FUNCTION_BLOCK T_ResultAggregate IMPLEMENTS I_ExecutionResult
VAR
	Results : ARRAY[0..ResultsUpperBound] OF I_ExecutionResult;
	Count   : UINT;
END_VAR
VAR CONSTANT
	ResultsUpperBound : UINT := 99;
END_VAR

METHOD Abort
VAR
    i      : DINT;
    Result : I_ExecutionResult;
    IP     : I_ListItem;
END_VAR
IF Count > 0 THEN
	FOR i := 0 TO Count - 1 DO
		Result := Results[i];
		IF Result <> 0 THEN
            Result.Abort(); 
        END_IF
    END_FOR
END_IF
END_METHOD

PROPERTY Aborted : BOOL
GET
VAR
    i      : UINT;
    Result : I_ExecutionResult;
END_VAR
Aborted := TRUE;
IF Count > 0 THEN
	FOR i := 0 TO Count - 1 DO
		Result := Results[i];
		IF Result <> 0 THEN
			Aborted := Aborted AND Result.Aborted; // Done if all result.aborted
		END_IF
	END_FOR
END_IF
END_GET
END_PROPERTY

PROPERTY Aborting : BOOL
GET
VAR
    i      : DINT;
    Result : I_ExecutionResult;
    IP     : I_ListItem;
END_VAR
Aborting := FALSE;
IF Count > 0 THEN
	FOR i := 0 TO Count - 1 DO
		Result := Results[i];
		IF Result <> 0 THEN
            Aborting := Aborting OR Result.Aborting; // Busy if any result.aborting
        END_IF
    END_FOR
END_IF
END_GET
END_PROPERTY

METHOD AddResult : BOOL
VAR_INPUT
	Result : I_ExecutionResult;
END_VAR
IF Count <= ResultsUpperBound THEN
	Results[Count] := Result;
	F_Inc(Count);
	AddResult := TRUE;
END_IF
END_METHOD

PROPERTY Busy : BOOL
GET
VAR
    i      : DINT;
    Result : I_ExecutionResult;
    IP     : I_ListItem;
END_VAR
Busy := FALSE;
IF Count > 0 THEN
	FOR i := 0 TO Count - 1 DO
		Result := Results[i];
		IF Result <> 0 THEN
            Busy := Busy OR Result.Busy; // Busy if any result.busy
        END_IF
    END_FOR
END_IF
END_GET
END_PROPERTY

METHOD Clear
VAR
    i      : UINT;
    Result : I_ExecutionResult;
END_VAR
IF Count > 0 THEN
    FOR i := 0 TO Count - 1 DO
		Result := Results[i];
		IF Result <> 0 THEN
			Result.Clear(); 
		END_IF
	END_FOR
END_IF

F_ClearMem(Results);
Count := 0;
END_METHOD

PROPERTY Done : BOOL
GET
VAR
    i      : DINT;
    Result : I_ExecutionResult;
    IP     : I_ListItem;
END_VAR
Done := TRUE;
IF Count > 0 THEN
	FOR i := 0 TO Count - 1 DO
		Result := Results[i];
		IF Result <> 0 THEN
			Done := Done AND Result.Done; // Done if all result.done
		END_IF
	END_FOR
END_IF
END_GET
END_PROPERTY

PROPERTY Error : BOOL
GET
VAR
    i      : DINT;
    Result : I_ExecutionResult;
    IP     : I_ListItem;
END_VAR
Error := FALSE;
IF Count > 0 THEN
	FOR i := 0 TO Count - 1 DO
		Result := Results[i];
		IF Result <> 0 THEN
			Error := Error OR Result.Error; // Error if any result.error
		END_IF
	END_FOR
END_IF
END_GET
END_PROPERTY

PROPERTY ErrorMsg : Tc2_System.T_MaxString
GET
VAR
    i      : DINT;
    Result : I_ExecutionResult;
    IP     : I_ListItem;
END_VAR
ErrorMsg := '';
IF Count > 0 THEN
	FOR i := 0 TO Count - 1 DO
		Result := Results[i];
		IF Result <> 0 THEN
			IF Result.Error THEN
				ErrorMsg := Result.ErrorMsg;
				RETURN;
			END_IF
		END_IF
	END_FOR
END_IF
END_GET
END_PROPERTY

PROPERTY Ready : BOOL
GET
VAR
    i      : DINT;
    Result : I_ExecutionResult;
    IP     : I_ListItem;
END_VAR
Ready := TRUE;
IF Count > 0 THEN
	FOR i := 0 TO Count - 1 DO
		Result := Results[i];
		IF Result <> 0 THEN
            Ready := Ready AND Result.Ready; // Ready if all result.ready
        END_IF
    END_FOR
END_IF
END_GET
END_PROPERTY

PROPERTY ResultCount : DINT
GET
ResultCount := Count;
END_GET
END_PROPERTY

PROPERTY Starting : BOOL
GET
VAR
    i      : DINT;
    Result : I_ExecutionResult;
    IP     : I_ListItem;
END_VAR
Starting := FALSE;
IF Count > 0 THEN
	FOR i := 0 TO Count - 1 DO
		Result := Results[i];
		IF Result <> 0 THEN
            Starting := Starting OR Result.Starting; // Starting if any result.starting
        END_IF
    END_FOR
END_IF
END_GET
END_PROPERTY

END_FUNCTION_BLOCK

(* stored: Version 1.1.0.1, ProductVersion 3.1.4024.15
   POU T_ResultAggregate: Id {454a147b-6226-4993-b56f-2debc6963635}, SpecialFunc None
   Folder Methods: Id {ec17c288-e510-45f8-8e37-6eb5b0058143}
   Folder Properties: Id {3d11f372-37c5-41b3-b352-a6a22277cfa1}
   Method Abort: Id {823e1046-db4f-4d09-9568-14fdd383baa5}
   Property Aborted: Id {acfc3263-0e48-4821-b470-e632d3592f91}
   Get Get: Id {089695a4-b523-4d4a-936a-6af96a3618ab}
   Property Aborting: Id {b62f2531-8180-4543-81d3-0b22b084b2f8}
   Get Get: Id {2f0cce7d-e42e-4e78-ab16-881c7500c8f4}
   Method AddResult: Id {a037aca6-2d76-47bb-ae65-f28ebca434dc}
   Property Busy: Id {4816830d-f3b9-42d1-8bce-e46a4f1ac9f0}
   Get Get: Id {bd41bfee-b27b-4e3a-ab02-258529323929}
   Method Clear: Id {df7f106c-b618-4f10-b8d6-6d0167d310bd}
   Property Done: Id {ac71d1f6-e94b-4b82-9737-80ef387eff14}
   Get Get: Id {c4bb208c-06a6-4f15-bd7e-21167842ac8a}
   Property Error: Id {4a084801-f1c2-4c69-a853-580e431dd29c}
   Get Get: Id {91812656-fd9e-4b5c-81cd-f800b7ec4a61}
   Property ErrorMsg: Id {27d8b087-df7b-4d80-9e54-086ef75e4c2e}
   Get Get: Id {3467fcda-438a-4236-b19a-6581ebd53bc0}
   Property Ready: Id {89a59524-360d-454d-95b9-1b5bfee550b1}
   Get Get: Id {cf43df40-3abf-4398-8c34-7437cb83dd24}
   Property ResultCount: Id {017d542d-7496-4360-9267-4e0033b3c085}
   Get Get: Id {4df98dac-690b-4072-bf68-703bf318d70d}
   Property Starting: Id {a9227d0a-cd83-4746-8b89-c559fb812990}
   Get Get: Id {2e0abc97-0bc7-417d-82b2-f39447040b3d} *)
